FUNCTION_BLOCK SM_AverageCurrent EXTENDS Current
VAR_INPUT
END_VAR
VAR_OUTPUT
END_VAR
VAR_IN_OUT
END_VAR
VAR
END_VAR

SUPER^();

END_FUNCTION_BLOCK

(* stored: Version 1.1.0.1, ProductVersion 3.1.4019.2
   POU SM_AverageCurrent: Id {a91ace93-9900-4ec3-bc8c-6997e3bd2549}, SpecialFunc None *)
